// TIA Portal V20 export
DATA_BLOCK "DB_HMI_PLC_Pos"   // DB135
// stored: InstanceOfName FB_HMI_PLC_Pos, InstanceOfType FB
"FB_HMI_PLC_Pos"
   // VAR_INPUT
   //    "HMI_Change Enable" : Bool;
   // END_VAR
   // VAR_IN_OUT
   //    ioPLC_State : Bool;
   //    ioHMI_State : Bool;
   // END_VAR
   // VAR
   //    PLC_StateMemo : Bool;
   //    HMI_StateMemo : Bool;
   // END_VAR
BEGIN
END_DATA_BLOCK
